INTERFACE I_ContainStatemachine EXTENDS I_Base

PROPERTY Statemachine : I_Statemachine
GET
END_GET
END_PROPERTY

END_INTERFACE

(* stored: Version 1.1.0.1, ProductVersion 3.1.4026.18
   Itf I_ContainStatemachine: Id {6e37caf7-1436-42b5-a1cf-f73ef666f192}
   Property Statemachine: Id {c58411a3-c15d-4915-a9cc-24d9901ced1b}
   Get Get: Id {dd204be9-35ef-45ea-ba65-68c12abe8039} *)
